FUNCTION_BLOCK fbDigitalOutput EXTENDS fbDigitalIO

METHOD PUBLIC Set
VAR_INPUT
	bValue : BOOL;
END_VAR
ioBIT := bValue;
END_METHOD

END_FUNCTION_BLOCK

(* stored: Version 1.1.0.1, ProductVersion 3.1.4024.15
   POU fbDigitalOutput: Id {c42d29ff-6d5a-47ff-94c8-15dae948f0bf}, SpecialFunc None
   Method Set: Id {c3a2d6d1-b8ed-43d5-8f12-d62b6d1998f7} *)
